TYPE ST_SawBladeData :
STRUCT
	rBladeDiameter : REAL;
	rBladeRadius : REAL;
	rBladeThickness: REAL;
	sBladeType : STRING;
END_STRUCT
END_TYPE

(* stored: Version 1.1.0.1
   DUT ST_SawBladeData: Id {cf847236-e954-45ee-8d69-0dd73122b276} *)
